// TwinCAT 3 PLC project SimulationPlc
// ProgramVersion: 3.1.4023.0
// libraries:
//   Tc2_Standard, * (Beckhoff Automation GmbH)
//   Tc2_System, * (Beckhoff Automation GmbH)
//   Tc3_Module, * (Beckhoff Automation GmbH)
// project tree:
//   POUs/ SimOven.TcPOU, SimRelay.TcPOU, MAIN.TcPOU
//   / SimulationTask.TcTTO
// real-time tasks:
//   TASK PlcTask: cycle T#10ms, priority 20, ADS port 350
//   TASK SimTask: cycle T#10ms, priority 1, ADS port 351
// variable links:
//   PLC/PLC Instance <-> SimulationPlc/SimulationPlc Instance
//     PlcTask Inputs/MAIN.oven.thermoCouple_Celcius <-> SimulationTask Outputs/MAIN.simOven.thermoCouple_Celcius
//     PlcTask Inputs/MAIN.relay.relayOnFeedback <-> SimulationTask Outputs/MAIN.simRelay.relayOnFeedback
//     PlcTask Outputs/MAIN.oven.heaterCurrent_Ampere <-> SimulationTask Inputs/MAIN.simOven.heaterCurrent_Ampere
//     PlcTask Outputs/MAIN.relay.turnOnRelay <-> SimulationTask Inputs/MAIN.simRelay.turnOnRelay

CONFIGURATION SimulationPlc
    RESOURCE PLC ON TwinCAT3
        TASK SimulationTask(INTERVAL := T#10ms, PRIORITY := 1);
        PROGRAM MAIN WITH SimulationTask : MAIN;
    END_RESOURCE
END_CONFIGURATION

// ---- POUs/MAIN.TcPOU
PROGRAM MAIN
VAR
    simRelay : SimRelay;
    simOven : SimOven;
END_VAR

simRelay();
simOven();

END_PROGRAM

// ---- POUs/SimRelay.TcPOU
FUNCTION_BLOCK SimRelay
VAR
    relayOnFeedback AT %Q* : BOOL;
    turnOnRelay AT %I* : BOOL;
    relayOnDelay : TON := (PT:=delay);
    relayOffDelay : TOF := (PT:=delay);
END_VAR
VAR CONSTANT
    delay : TIME := T#1S;
END_VAR

relayOnDelay(IN:=turnOnRelay);
IF relayOnDelay.Q THEN
    relayOnFeedback := TRUE;
END_IF

relayOffDelay(IN:=turnOnRelay);
IF NOT relayOffDelay.Q THEN
    relayOnFeedback := FALSE;
END_IF

END_FUNCTION_BLOCK

// ---- POUs/SimOven.TcPOU
FUNCTION_BLOCK SimOven
VAR
    thermoCouple_Celcius AT %Q* : REAL;
    heaterCurrent_Ampere AT %I* : REAL;
END_VAR
VAR
    previousTemperature : REAL;
    filterParameter : REAL := 0.995;
END_VAR

thermoCouple_Celcius := previousTemperature * filterParameter
    + LIMIT(20, TO_REAL(EXPT(heaterCurrent_Ampere, 2)), 1E5) * (1 - filterParameter);
previousTemperature := thermoCouple_Celcius;

END_FUNCTION_BLOCK
